FUNCTION_BLOCK StringValue_AIWS (* Input service interface function block for wide string input data *)
  (* Description: Copyright (c) 2026 HR Agrartechnik GmbH This program and the accompanying materials are made available under the terms of the Eclipse Public License 2.0 which is available at https://www.eclipse.org/legal/epl-2.0/ SPDX-License-Identifier: EPL-2.0 *)
  (* Version 1.0, 2026-04-13, Franz Höpfinger, HR Agrartechnik GmbH *)
  PACKAGE isobus::UT::io::StringValue;
  IMPORT eclipse4diac::core::TypeHash;
  IMPORT isobus::UT::Q::const::IDs::ID_NULL;
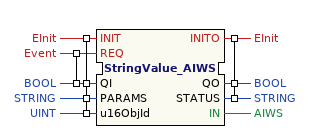
  EVENT_INPUT
    INIT : EInit WITH QI, PARAMS, u16ObjId; (* Service Initialization *)
    REQ WITH QI; (* Service Request *)
  END_EVENT
  EVENT_OUTPUT
    INITO : EInit WITH QO, STATUS; (* Initialization Confirm *)
  END_EVENT
  VAR_INPUT
    QI : BOOL; (* Event Input Qualifier *)
    PARAMS : STRING; (* Service Parameters *)
    u16ObjId : UINT := ID_NULL; (* Object ID *)
  END_VAR
  VAR_OUTPUT
    QO : BOOL; (* Event Output Qualifier *)
    STATUS : STRING; (* Service Status *)
  END_VAR
  PLUGS
    IN : adapter::types::unidirectional::AIWS; (* Input data from resource *)
  END_PLUGS
  FBS
    StringValue_IWS : isobus::UT::io::StringValue::StringValue_IWS;
  END_FBS
  EVENT_CONNECTIONS
    INIT TO StringValue_IWS.INIT;
    REQ TO StringValue_IWS.REQ;
    StringValue_IWS.IND TO IN.E1;
    StringValue_IWS.CNF TO IN.E1;
    StringValue_IWS.INITO TO INITO;
  END_CONNECTIONS
  DATA_CONNECTIONS
    QI TO StringValue_IWS.QI;
    PARAMS TO StringValue_IWS.PARAMS;
    u16ObjId TO StringValue_IWS.u16ObjId;
    StringValue_IWS.IN TO IN.D1;
    StringValue_IWS.STATUS TO STATUS;
    StringValue_IWS.QO TO QO;
  END_CONNECTIONS
END_FUNCTION_BLOCK
